// TIA Portal V16 export
// export: Created 2021-07-12T14:47:03.3757701Z, ExportSetting WithDefaults, DisplayName Totally Integrated Automation Portal, DisplayVersion V16, DisplayName TIA Portal Version Control Interface, DisplayVersion V16, DisplayName TIA Portal Openness, DisplayVersion V16, DisplayName STEP 7 Professional, DisplayVersion V16, DisplayName STEP 7 Safety, DisplayVersion V16, DisplayName WinCC Professional, DisplayVersion V16
FUNCTION_BLOCK "LSimaHydTO_ValvesControl"   // FB33004, LAD
TITLE = LSimaHydTO_ValvesControl
{ S7_Optimized_Access := 'TRUE' }
AUTHOR : APC_ERLF
FAMILY : LSimaHydTO
VERSION : 1.0
// //============================================================================
// //SIEMENS AG // (c)Copyright 2019 All Rights Reserved
// //--------------------------------------------------------------------------------
// //Library:       LSimaHydTO
// //Tested with:   S7-15xx
// //Engineering:   TIA Portal  V15
// //Restrictions:  -
// //Requirements:  S7-1500 (FW 2.5)
// //Functionality: - for internal use
// //
// //--------------------------------------------------------------------------------
// //Change log table:
// //
// //Version     Date          Expert in charge    Changes applied
// //01.00.00    15.03.2018    APC_ERLF            First released version
// //============================================================================
// stored: AutoNumber true, IsIECCheckEnabled false, IsRetainMemResEnabled false, MemoryReserve 0, SetENOAutomatically false, UDAEnableTagReadback false
   VAR_INPUT
      enable { ExternalAccessible := 'False'; ExternalVisible := 'False'; ExternalWritable := 'False'} : Bool;
      reqForward { ExternalAccessible := 'False'; ExternalVisible := 'False'; ExternalWritable := 'False'} : Bool;
      reqBackward { ExternalAccessible := 'False'; ExternalVisible := 'False'; ExternalWritable := 'False'} : Bool;
      sampleTime { ExternalAccessible := 'False'; ExternalVisible := 'False'; ExternalWritable := 'False'} : LReal;   // cycle time of synchronous OB [s]
   END_VAR
   VAR_OUTPUT
      rampingForward { ExternalAccessible := 'False'; ExternalVisible := 'False'; ExternalWritable := 'False'} : Bool;   // enable signal for ramping in positive direction
      rampingBackward { ExternalAccessible := 'False'; ExternalVisible := 'False'; ExternalWritable := 'False'} : Bool;   // enable signal for ramping in negative direction
   END_VAR
   VAR_IN_OUT
      axisData : "LSimaHydTO_typeAxisData";   // Axis data
   END_VAR
   VAR
      instTOFChangeDir { ExternalAccessible := 'False'; ExternalVisible := 'False'; ExternalWritable := 'False'; S7_SetPoint := 'True'} : "LSimaHydTO_TOF_Cycl";
      statChangeDirEnabled { ExternalAccessible := 'False'; ExternalVisible := 'False'; ExternalWritable := 'False'} : Bool;
      statSRForward { ExternalAccessible := 'False'; ExternalVisible := 'False'; ExternalWritable := 'False'} : Bool;
      statReqForward { ExternalAccessible := 'False'; ExternalVisible := 'False'; ExternalWritable := 'False'} : Bool;
      instTONValveForward { ExternalAccessible := 'False'; ExternalVisible := 'False'; ExternalWritable := 'False'; S7_SetPoint := 'True'} : "LSimaHydTO_TON_Cycl";
      statReqBackward { ExternalAccessible := 'False'; ExternalVisible := 'False'; ExternalWritable := 'False'} : Bool;
      statSRBackward { ExternalAccessible := 'False'; ExternalVisible := 'False'; ExternalWritable := 'False'} : Bool;
      instTONValveBackward { ExternalAccessible := 'False'; ExternalVisible := 'False'; ExternalWritable := 'False'; S7_SetPoint := 'True'} : "LSimaHydTO_TON_Cycl";
   END_VAR
   VAR_TEMP
      tempLreal : LReal;
   END_VAR
   VAR_TEMP   // added for the SCL form of the ladder/FBD networks
      _w1 : Bool;
   END_VAR
BEGIN

REGION Network 1: the max. safety position was passed
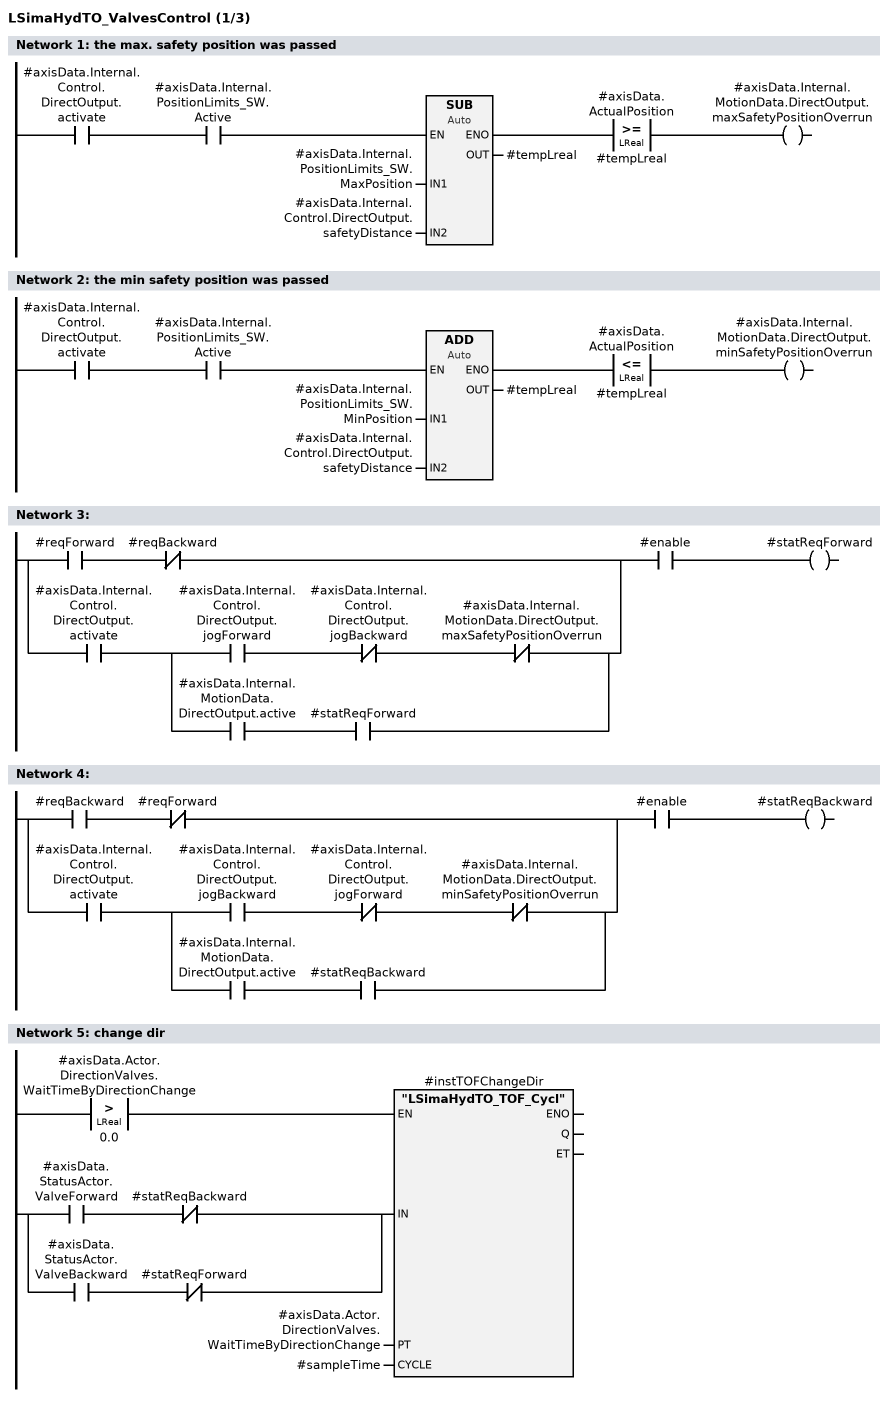
   RUNG wire#powerrail
      Contact( #axisData.Internal.Control.DirectOutput.activate )
      Contact( #axisData.Internal.PositionLimits_SW.Active )
      Sub(in1 := #axisData.Internal.PositionLimits_SW.MaxPosition, in2 := #axisData.Internal.Control.DirectOutput.safetyDistance, out => #tempLreal)
      { S7_Templates := "SrcType := LReal" } GE_Contact(in1 := #axisData.ActualPosition, in2 := #tempLreal)
      Coil( #axisData.Internal.MotionData.DirectOutput.maxSafetyPositionOverrun )
   END_RUNG
   // the same network as SCL:
   #_w1 := #axisData.Internal.Control.DirectOutput.activate AND #axisData.Internal.PositionLimits_SW.Active;
   IF #_w1 THEN
       #tempLreal := #axisData.Internal.PositionLimits_SW.MaxPosition - #axisData.Internal.Control.DirectOutput.safetyDistance;
   END_IF;
   #axisData.Internal.MotionData.DirectOutput.maxSafetyPositionOverrun := #_w1 AND (#axisData.ActualPosition >= #tempLreal);
END_REGION

REGION Network 2: the min safety position was passed
   RUNG wire#powerrail
      Contact( #axisData.Internal.Control.DirectOutput.activate )
      Contact( #axisData.Internal.PositionLimits_SW.Active )
      Add(in1 := #axisData.Internal.PositionLimits_SW.MinPosition, in2 := #axisData.Internal.Control.DirectOutput.safetyDistance, out => #tempLreal)
      { S7_Templates := "SrcType := LReal" } LE_Contact(in1 := #axisData.ActualPosition, in2 := #tempLreal)
      Coil( #axisData.Internal.MotionData.DirectOutput.minSafetyPositionOverrun )
   END_RUNG
   // the same network as SCL:
   #_w1 := #axisData.Internal.Control.DirectOutput.activate AND #axisData.Internal.PositionLimits_SW.Active;
   IF #_w1 THEN
       #tempLreal := #axisData.Internal.PositionLimits_SW.MinPosition + #axisData.Internal.Control.DirectOutput.safetyDistance;
   END_IF;
   #axisData.Internal.MotionData.DirectOutput.minSafetyPositionOverrun := #_w1 AND (#axisData.ActualPosition <= #tempLreal);
END_REGION

REGION Network 3
   RUNG wire#powerrail
      Contact( #reqForward )
      I_Contact( #reqBackward )
      wire#w1
      Contact( #enable )
      Coil( #statReqForward )
   END_RUNG
   RUNG wire#powerrail
      Contact( #axisData.Internal.Control.DirectOutput.activate )
      wire#w2
      Contact( #axisData.Internal.Control.DirectOutput.jogForward )
      I_Contact( #axisData.Internal.Control.DirectOutput.jogBackward )
      I_Contact( #axisData.Internal.MotionData.DirectOutput.maxSafetyPositionOverrun )
   END_RUNG wire#w1
   RUNG wire#w2
      Contact( #axisData.Internal.MotionData.DirectOutput.active )
      Contact( #statReqForward )
   END_RUNG wire#w1
   // the same network as SCL:
   #statReqForward := ((#reqForward AND NOT #reqBackward) OR (#axisData.Internal.Control.DirectOutput.activate AND ((#axisData.Internal.Control.DirectOutput.jogForward AND NOT #axisData.Internal.Control.DirectOutput.jogBackward AND NOT #axisData.Internal.MotionData.DirectOutput.maxSafetyPositionOverrun) OR (#axisData.Internal.MotionData.DirectOutput.active AND #statReqForward)))) AND #enable;
END_REGION

REGION Network 4
   RUNG wire#powerrail
      Contact( #reqBackward )
      I_Contact( #reqForward )
      wire#w1
      Contact( #enable )
      Coil( #statReqBackward )
   END_RUNG
   RUNG wire#powerrail
      Contact( #axisData.Internal.Control.DirectOutput.activate )
      wire#w2
      Contact( #axisData.Internal.Control.DirectOutput.jogBackward )
      I_Contact( #axisData.Internal.Control.DirectOutput.jogForward )
      I_Contact( #axisData.Internal.MotionData.DirectOutput.minSafetyPositionOverrun )
   END_RUNG wire#w1
   RUNG wire#w2
      Contact( #axisData.Internal.MotionData.DirectOutput.active )
      Contact( #statReqBackward )
   END_RUNG wire#w1
   // the same network as SCL:
   #statReqBackward := ((#reqBackward AND NOT #reqForward) OR (#axisData.Internal.Control.DirectOutput.activate AND ((#axisData.Internal.Control.DirectOutput.jogBackward AND NOT #axisData.Internal.Control.DirectOutput.jogForward AND NOT #axisData.Internal.MotionData.DirectOutput.minSafetyPositionOverrun) OR (#axisData.Internal.MotionData.DirectOutput.active AND #statReqBackward)))) AND #enable;
END_REGION

REGION Network 5: change dir
   RUNG wire#powerrail
      { S7_Templates := "SrcType := LReal" } GT_Contact(in1 := #axisData.Actor.DirectionValves.WaitTimeByDirectionChange, in2 := 0.0)
      #instTOFChangeDir(IN := wire#w1, PT := #axisData.Actor.DirectionValves.WaitTimeByDirectionChange, CYCLE := #sampleTime, Q =>, ET =>)
   END_RUNG
   RUNG wire#powerrail
      Contact( #axisData.StatusActor.ValveForward )
      I_Contact( #statReqBackward )
   END_RUNG wire#w1
   RUNG wire#powerrail
      Contact( #axisData.StatusActor.ValveBackward )
      I_Contact( #statReqForward )
   END_RUNG wire#w1
   // the same network as SCL:
   IF #axisData.Actor.DirectionValves.WaitTimeByDirectionChange > 0.0 THEN
       #instTOFChangeDir(IN := (#axisData.StatusActor.ValveForward AND NOT #statReqBackward) OR (#axisData.StatusActor.ValveBackward AND NOT #statReqForward),   // "LSimaHydTO_TOF_Cycl"
                         PT := #axisData.Actor.DirectionValves.WaitTimeByDirectionChange,
                         CYCLE := #sampleTime);
   END_IF;
END_REGION

REGION Network 6
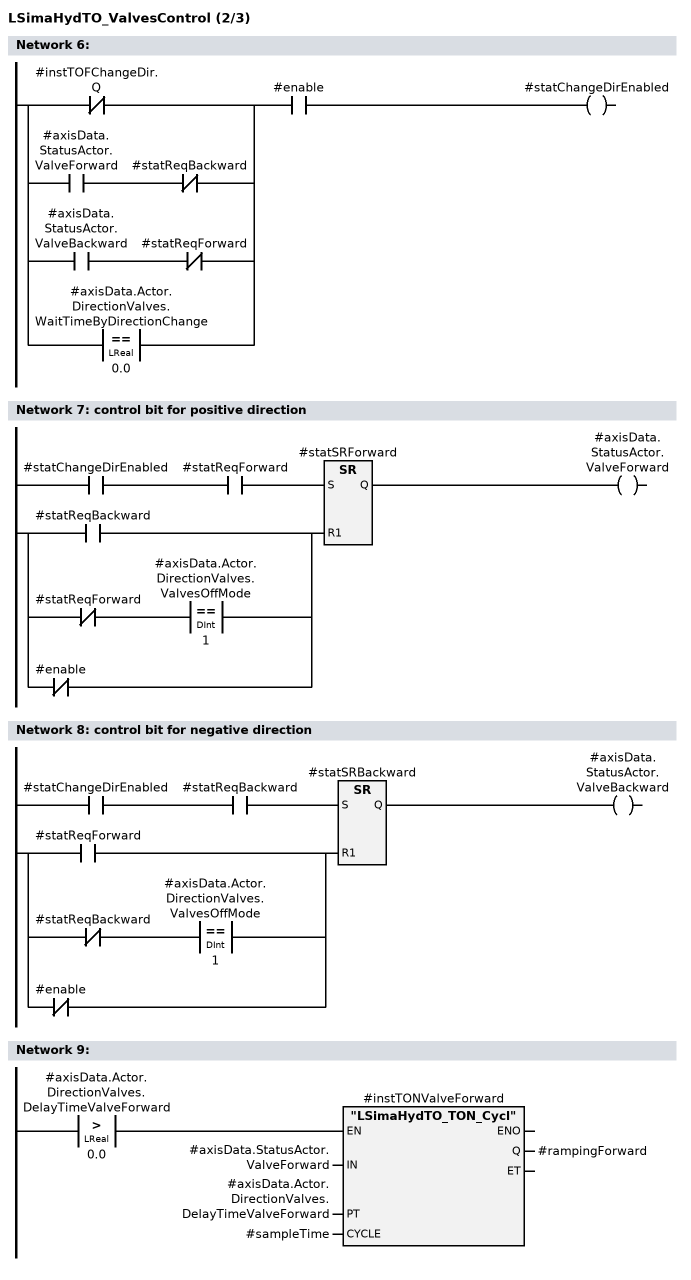
   RUNG wire#powerrail
      I_Contact( #instTOFChangeDir.Q )
      wire#w1
      Contact( #enable )
      Coil( #statChangeDirEnabled )
   END_RUNG
   RUNG wire#powerrail
      Contact( #axisData.StatusActor.ValveForward )
      I_Contact( #statReqBackward )
   END_RUNG wire#w1
   RUNG wire#powerrail
      Contact( #axisData.StatusActor.ValveBackward )
      I_Contact( #statReqForward )
   END_RUNG wire#w1
   RUNG wire#powerrail
      { S7_Templates := "SrcType := LReal" } EQ_Contact(in1 := #axisData.Actor.DirectionValves.WaitTimeByDirectionChange, in2 := 0.0)
   END_RUNG wire#w1
   // the same network as SCL:
   #statChangeDirEnabled := (NOT #instTOFChangeDir.Q OR (#axisData.StatusActor.ValveForward AND NOT #statReqBackward) OR (#axisData.StatusActor.ValveBackward AND NOT #statReqForward) OR (#axisData.Actor.DirectionValves.WaitTimeByDirectionChange = 0.0)) AND #enable;
END_REGION

REGION Network 7: control bit for positive direction
   RUNG wire#powerrail
      Contact( #statChangeDirEnabled )
      Contact( #statReqForward )
      S_SR(operand := #statSRForward, r1 := wire#w1)
      Coil( #axisData.StatusActor.ValveForward )
   END_RUNG
   RUNG wire#powerrail
      Contact( #statReqBackward )
   END_RUNG wire#w1
   RUNG wire#powerrail
      I_Contact( #statReqForward )
      { S7_Templates := "SrcType := DInt" } EQ_Contact(in1 := #axisData.Actor.DirectionValves.ValvesOffMode, in2 := 1)
   END_RUNG wire#w1
   RUNG wire#powerrail
      I_Contact( #enable )
   END_RUNG wire#w1
   // the same network as SCL:
   IF #statChangeDirEnabled AND #statReqForward THEN
       #statSRForward := TRUE;   // SR flip-flop
   END_IF;
   IF #statReqBackward OR (NOT #statReqForward AND (#axisData.Actor.DirectionValves.ValvesOffMode = 1)) OR NOT #enable THEN
       #statSRForward := FALSE;
   END_IF;
   #axisData.StatusActor.ValveForward := #statSRForward;
END_REGION

REGION Network 8: control bit for negative direction
   RUNG wire#powerrail
      Contact( #statChangeDirEnabled )
      Contact( #statReqBackward )
      S_SR(operand := #statSRBackward, r1 := wire#w1)
      Coil( #axisData.StatusActor.ValveBackward )
   END_RUNG
   RUNG wire#powerrail
      Contact( #statReqForward )
   END_RUNG wire#w1
   RUNG wire#powerrail
      I_Contact( #statReqBackward )
      { S7_Templates := "SrcType := DInt" } EQ_Contact(in1 := #axisData.Actor.DirectionValves.ValvesOffMode, in2 := 1)
   END_RUNG wire#w1
   RUNG wire#powerrail
      I_Contact( #enable )
   END_RUNG wire#w1
   // the same network as SCL:
   IF #statChangeDirEnabled AND #statReqBackward THEN
       #statSRBackward := TRUE;   // SR flip-flop
   END_IF;
   IF #statReqForward OR (NOT #statReqBackward AND (#axisData.Actor.DirectionValves.ValvesOffMode = 1)) OR NOT #enable THEN
       #statSRBackward := FALSE;
   END_IF;
   #axisData.StatusActor.ValveBackward := #statSRBackward;
END_REGION

REGION Network 9
   RUNG wire#powerrail
      { S7_Templates := "SrcType := LReal" } GT_Contact(in1 := #axisData.Actor.DirectionValves.DelayTimeValveForward, in2 := 0.0)
      #instTONValveForward(IN := #axisData.StatusActor.ValveForward, PT := #axisData.Actor.DirectionValves.DelayTimeValveForward, CYCLE := #sampleTime, Q => #rampingForward, ET =>)
   END_RUNG
   // the same network as SCL:
   IF #axisData.Actor.DirectionValves.DelayTimeValveForward > 0.0 THEN
       #instTONValveForward(IN := #axisData.StatusActor.ValveForward,   // "LSimaHydTO_TON_Cycl"
                            PT := #axisData.Actor.DirectionValves.DelayTimeValveForward,
                            CYCLE := #sampleTime,
                            Q => #rampingForward);
   END_IF;
END_REGION

REGION Network 10: enable signal for ramping in positive direction
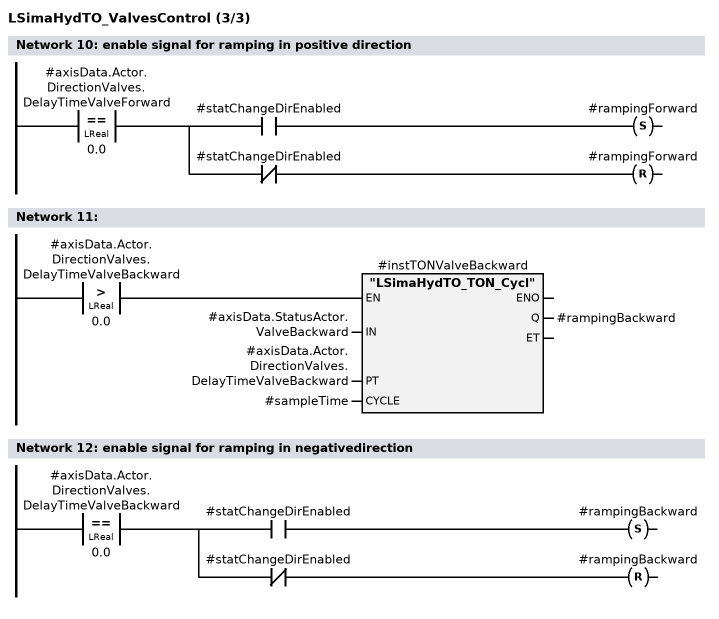
   RUNG wire#powerrail
      { S7_Templates := "SrcType := LReal" } EQ_Contact(in1 := #axisData.Actor.DirectionValves.DelayTimeValveForward, in2 := 0.0)
      wire#w1
      Contact( #statChangeDirEnabled )
      S_Coil( #rampingForward )
   END_RUNG
   RUNG wire#w1
      I_Contact( #statChangeDirEnabled )
      R_Coil( #rampingForward )
   END_RUNG
   // the same network as SCL:
   #_w1 := #axisData.Actor.DirectionValves.DelayTimeValveForward = 0.0;
   IF #_w1 AND #statChangeDirEnabled THEN #rampingForward := TRUE; END_IF;
   IF #_w1 AND NOT #statChangeDirEnabled THEN #rampingForward := FALSE; END_IF;
END_REGION

REGION Network 11
   RUNG wire#powerrail
      { S7_Templates := "SrcType := LReal" } GT_Contact(in1 := #axisData.Actor.DirectionValves.DelayTimeValveBackward, in2 := 0.0)
      #instTONValveBackward(IN := #axisData.StatusActor.ValveBackward, PT := #axisData.Actor.DirectionValves.DelayTimeValveBackward, CYCLE := #sampleTime, Q => #rampingBackward, ET =>)
   END_RUNG
   // the same network as SCL:
   IF #axisData.Actor.DirectionValves.DelayTimeValveBackward > 0.0 THEN
       #instTONValveBackward(IN := #axisData.StatusActor.ValveBackward,   // "LSimaHydTO_TON_Cycl"
                             PT := #axisData.Actor.DirectionValves.DelayTimeValveBackward,
                             CYCLE := #sampleTime,
                             Q => #rampingBackward);
   END_IF;
END_REGION

REGION Network 12: enable signal for ramping in negativedirection
   RUNG wire#powerrail
      { S7_Templates := "SrcType := LReal" } EQ_Contact(in1 := #axisData.Actor.DirectionValves.DelayTimeValveBackward, in2 := 0.0)
      wire#w1
      Contact( #statChangeDirEnabled )
      S_Coil( #rampingBackward )
   END_RUNG
   RUNG wire#w1
      I_Contact( #statChangeDirEnabled )
      R_Coil( #rampingBackward )
   END_RUNG
   // the same network as SCL:
   #_w1 := #axisData.Actor.DirectionValves.DelayTimeValveBackward = 0.0;
   IF #_w1 AND #statChangeDirEnabled THEN #rampingBackward := TRUE; END_IF;
   IF #_w1 AND NOT #statChangeDirEnabled THEN #rampingBackward := FALSE; END_IF;
END_REGION
END_FUNCTION_BLOCK
